(* PLC project Generated.project, CODESYS CODESYS V3.5 SP19 Patch 1 *)
(* stored: creationDateTime 2026-08-18T01:51:35.943984, modificationDateTime 2026-08-18T01:51:35.943984 *)

(* values of E_CycleStep: X0_PREPARATION: Début de graphe : à la TRÉMIE, treuils en position HAUTE; X1_HOMING: Vitesses lentes pour chercher capteur top + référencement; X2_WORK_POS_SELECT: Sélection cible Trémie/P1/Maintenance + translation validée; X3_OPEN_BUCKET: Ouverture benne (si déjà ouverte -> passe vite); X4_DESCEND_OPEN: Plongée benne ouverte, M1+M2 synchro, Kobold mesure ON; X5_BOTTOM_CONFIRMED: Fond validé (FB_DiveSearch) ; arrêt descente; X6_CLOSE_BUCKET: Fermeture benne — tolérance « à peu près fermé »; X7_CTRL_ASCENT: Remontée palier 1 de contrôle; X8_ASCENT_LOADED: Remontée nominale jusqu'à limite haute; X9_DRAIN_PAUSE: Égouttage temporisé — temps affiché IHM; X10_TRANSLATE_DUMP: Translation vers trémie + avertissements IHM; X11_OPEN_DUMP: Ouverture benne = vidage ; montée possible, descente ouvre; X13_DONE_SYNC: Fin de cycle, synchronisation finale (R4) + compteur; STABILIZING: État d'attente/stabilisation — pas une erreur *)

{attribute 'qualified_only'}
{attribute 'strict'}
TYPE E_CycleStep : (X0_PREPARATION := 0, X1_HOMING := 1, X2_WORK_POS_SELECT := 2, X3_OPEN_BUCKET := 3, X4_DESCEND_OPEN := 4, X5_BOTTOM_CONFIRMED := 5, X6_CLOSE_BUCKET := 6, X7_CTRL_ASCENT := 7, X8_ASCENT_LOADED := 8, X9_DRAIN_PAUSE := 9, X10_TRANSLATE_DUMP := 10, X11_OPEN_DUMP := 11, X13_DONE_SYNC := 13, STABILIZING := 14);
END_TYPE
